INTERFACE ITrackCtrl

METHOD ComputeNextPos : BOOL
VAR_INPUT
END_VAR

VAR_OUTPUT
	newPos : LREAL;
END_VAR
END_METHOD

METHOD HandleStates : BOOL
VAR_INPUT
END_VAR
END_METHOD

METHOD Init : BOOL
VAR_INPUT
END_VAR
END_METHOD

METHOD IsError : BOOL
VAR_INPUT
END_VAR
END_METHOD

METHOD MoveInPos : BOOL
VAR_INPUT
	refMotion: REFERENCE TO T_MOTOR_MOTION;
END_VAR
END_METHOD

METHOD MoveInSpeed
VAR_INPUT
	refMotion: REFERENCE TO T_MOTOR_MOTION;
END_VAR
END_METHOD

METHOD Reset : BOOL
VAR_INPUT
END_VAR
END_METHOD

END_INTERFACE

(* stored: Version 1.1.0.1, ProductVersion 3.1.4022.9
   Itf ITrackCtrl: Id {190bd2ba-4f1b-43d1-8419-d9931b546093}
   Method ComputeNextPos: Id {7d0345c5-5e48-4eb5-aa71-1c7a122fd260}
   Method HandleStates: Id {b7501932-62ac-479b-af6b-4e1e30081d16}
   Method Init: Id {adfd036f-4226-4e75-9683-67c191735e72}
   Method IsError: Id {7ffa8d83-850f-49dc-8bcb-be1f45946c39}
   Method MoveInPos: Id {ab22d95d-e8d4-4c69-88cd-1392bbcd8759}
   Method MoveInSpeed: Id {c914b374-d828-4404-b57c-98b4b8a5551d}
   Method Reset: Id {5c95606e-71cf-451e-afbc-1b9795aac039} *)
